FUNCTION_BLOCK FB_AnnealingOven
VAR_INPUT
END_VAR
VAR_OUTPUT
	bStatusOn_ExhaustGas : BOOL;
	bStatusOn_Sealing : BOOL;
END_VAR
VAR
	//modbus tcp communication
	ModbusReader : FB_MBReadRegs;
	aModbus : ARRAY  [0..61] OF WORD;
	bReadModbus	: BOOL := FALSE;
	bStartTimer : BOOL;
	Timer : TON;
END_VAR

Timer(IN := bStartTimer,
	PT := T#2S);
	
bStartTimer := TRUE;
IF Timer.Q THEN
	bReadModbus := TRUE;
	bStartTimer := FALSE;	
END_IF

ModbusReader(sIPAddr := GlobalVariables.sIP_Annealing_Oven,
	nTCPPort := 502,
	nUnitID := 255,
	nQuantity := 80,
	nMBAddr := 800,
	cbLength := 122,
	pDestAddr := ADR(aModbus),
	bExecute := bReadModbus,
	tTimeout  := T#20S);
bReadModbus := FALSE;

bStatusOn_ExhaustGas := FALSE;
bStatusOn_Sealing := FALSE;

END_FUNCTION_BLOCK

(* stored: Version 1.1.0.1, ProductVersion 3.1.4024.10
   POU FB_AnnealingOven: Id {9d60a342-9fa8-4850-9da6-ab1de2c9e1f5}, SpecialFunc None *)
